FUNCTION_BLOCK TcoCvirII EXTENDS TcoCore.TcoComponent IMPLEMENTS ITcoScrewdriver //TODO: EXTENDS TcoIo.TcoPnIoComponent //IMPLEMENTS TcoAbstractions.ITcoScrewdriver
VAR_IN_OUT
	inoIoData : TcoCvirII_Io;
END_VAR

VAR
	_config : TcoCvirII_Config;
	_status : TcoCvirII_Status;
END_VAR

VAR
	_data : TcoCvirII_Data;
	_results : TcoCvirII_Results;
	
	_state : TcoCore.TcoState(THIS^, eRestoreMode.None);
	
	{attribute 'hide'}
	_timer : TON;

	//INPUT VARIABLES	
	{attribute addProperty Name "<#Screwing Program Number#>"}
	_programNo : BYTE;
	{attribute addProperty Name "<#Automatic Start#>"}
	_automaticStart : BOOL;
	
	{attribute addProperty Name "<#Run screwing cycle#>"}
	_screwingTask : TcoCore.TcoTask(THIS^);					//sequence
	
//	{attribute addProperty Name "<#Screwing program number#>"}	
//	_programNumber : BYTE; 
	{attribute addProperty Name "<#Set screwing program#>"}
	_setScrewingProgramTask : TcoCore.TcoTask(THIS^); 		//waiting for hw response
	
	{attribute addProperty Name "<#Enable#>"}
	_enableTask : TcoCore.TcoTask(THIS^);					//immediately done
	{attribute addProperty Name "<#Disable#>"}
	_disableTask : TcoCore.TcoTask(THIS^);
	{attribute addProperty Name "<#Forward#>"}
	_forwardTask : TcoCore.TcoTask(THIS^);					//sequence
	{attribute addProperty Name "<#Reverse#>"}
	_reverseTask : TcoCore.TcoTask(THIS^);					//sequence
	{attribute addProperty Name "<#Restore#>"}
    _restoreTask : TcoCore.TcoTask(THIS^);
END_VAR

VAR
    {attribute 'hide'} 
	_varInfo : __SYSTEM.VAR_INFO;
    {attribute 'hide'} 
	_sb : TcoCore.StringBuilder;
END_VAR

IF InvalidReference() THEN
    RETURN;
END_IF

//SUPER^(inPnIoBoxState := THIS^.inoIoData.PnIoBoxState, inPnIoBoxDiag := THIS^.inoIoData.PnIoBoxDiag);

InitializeComponent();

//IF NOT SUPER^.ProfinetReady THEN
//	THIS^._status.ActionDescription := '<#Not ready for operation by means of Profinet network!#>';	
//END_IF

//IF SUPER^.ProfinetReady AND THIS^._status.ActionDescription = '<#Not ready for operation by means of Profinet network!#>' THEN
//	THIS^._status.ActionDescription := '<#Ready for operation!#>';	
//END_IF

//*************RESTORE********************
_restoreTask.Enabled := TRUE;
IF _restoreTask.Execute() THEN
	Restore();
END_IF
//****************************************

//**********SET SCREWING PROGRAM**********
_setScrewingProgramTask.Enabled := TRUE;
IF _setScrewingProgramTask.Execute() THEN
	_data.ScrewingProgramOUT := _programNo;
	IF (_data.ScrewingProgramOUT  = _data.ScrewingProgramIN) THEN
		_setScrewingProgramTask.DoneWhen(TRUE);
	END_IF
END_IF
//****************************************

//****************SCREWING****************
_screwingTask.Enabled := NOT _forwardTask.Busy AND NOT _reverseTask.Busy;
IF _screwingTask.Execute() THEN
	_screwingTask.DoneWhen(ScrewingInternal());
END_IF
//****************************************

//****************ENABLE******************
_enableTask.Enabled := TRUE;
IF _enableTask.Execute() THEN
	_data.Control.SpindleValidation := TRUE;
	_enableTask.DoneWhen(TRUE);
END_IF
//****************************************

//****************DISABLE******************
_disableTask.Enabled := TRUE;
IF _disableTask.Execute() THEN
	_data.Control.SpindleValidation := FALSE;
	_disableTask.DoneWhen(TRUE);
END_IF
//*****************************************

//****************FORWARD******************
_forwardTask.Enabled := NOT _screwingTask.Busy AND NOT _reverseTask.Busy;
IF _forwardTask.Execute() THEN
	_forwardTask.DoneWhen(ScrewClockwiseInternal());
END_IF
//*****************************************

//****************REVERSE******************
_reverseTask.Enabled := NOT _screwingTask.Busy AND NOT _forwardTask.Busy;
IF _reverseTask.Execute() THEN
	_reverseTask.DoneWhen(ScrewCounterClockwiseInternal());
END_IF
//*****************************************

(*~
	<docu>
		<summary>
			Gets the configuration of the screwdriver. 					
		</summary>			
	</docu>	
~*)
PROPERTY Config : REFERENCE TO TcoCvirII_Config
GET
Config REF= _config;
END_GET
END_PROPERTY

PROPERTY DisableTask : TcoCore.ITcoTaskStatus
GET
DisableTask := THIS^._disableTask;
END_GET
END_PROPERTY

PROPERTY EnableTask : TcoCore.ITcoTaskStatus
GET
EnableTask := THIS^._enableTask;
END_GET
END_PROPERTY

PROPERTY ForwardTask : TcoCore.ITcoTaskStatus
GET
ForwardTask := THIS^._forwardTask;
END_GET
END_PROPERTY

METHOD PRIVATE InitializeComponent
VAR_INPUT
END_VAR
IF(InvalidReference()) THEN
	RETURN;
END_IF

//Reading input data
_data.Status.CycleBit1 := inoIoData.Status.0;
_data.Status.CycleBit2 := inoIoData.Status.1;
_data.Status.CycleBit4 := inoIoData.Status.2;
_data.Status.Ready := inoIoData.Status.3;
_data.Status.InCycle := inoIoData.Status.4;
_data.Status.Passed := inoIoData.Status.5;
_data.Status.Failed := inoIoData.Status.6;
_data.Status.NumberOfCyclesOk := inoIoData.Status.7;

_data.ScrewingProgramIN := inoIoData.ScrewingProgramIN;

_data.Torque := inoIoData.Torque;
_data.TorqueTrend := inoIoData.TorqueTrend;
_data.Angle := inoIoData.Angle;
_data.AngleTrend := inoIoData.AngleTrend;


//Write output data
inoIoData.Control.0 := _data.Control.CycleBit1;
inoIoData.Control.1 := _data.Control.CycleBit2;
inoIoData.Control.2 := _data.Control.CycleBit4;
inoIoData.Control.3 := _data.Control.SpindleValidation;
inoIoData.Control.4 := _data.Control.ErrorAck;
inoIoData.Control.5 := _data.Control.StartCycle;
inoIoData.Control.6 := _data.Control.Direction;
inoIoData.Control.7 := _data.Control.Reset;

inoIoData.ScrewingProgramOUT := _data.ScrewingProgramOUT;
END_METHOD

METHOD INTERNAL InvalidReference : BOOL
InvalidReference := FALSE;
IF NOT __ISVALIDREF(inoIoData) THEN
	_varInfo :=__VARINFO(inoIoData);
	Messenger.Error(_sb.Clear().Append('<#Invalid reference: #>').Append(_varInfo.Symbol).ToString());
    InvalidReference := TRUE;
END_IF
END_METHOD

(*~
	<docu>
		<summary>
			Restores this instance to the Ready state. Can be called explicitly or from within one of the restore mechanisms.	
		</summary>			
	</docu>	
~*)
METHOD  Restore : ITcoRestorable
_screwingTask.Restore();
_setScrewingProgramTask.Restore();

_enableTask.Restore();
_disableTask.Restore();

_forwardTask.Restore();
_reverseTask.Restore();

_state.Restore();

THIS^._results.Torque := 0;
THIS^._results.TorqueTrend := 0;
THIS^._results.Angle := 0;
THIS^._results.AngleTrend := 0;
	
IF InvalidReference() THEN
    RETURN;
END_IF

Tc2_System.MEMSET(destAddr:= ADR(THIS^.inoIoData) , fillByte:= 0 , n:= SIZEOF(THIS^.inoIoData));

_status.ActionDescription := '<#Restore executed!#>';
_restoreTask.Restore();
END_METHOD

PROPERTY Results : TcoCvirII_Results
GET
Results := _results;
END_GET
END_PROPERTY

PROPERTY ReverseTask : TcoCore.ITcoTaskStatus
GET
ReverseTask := THIS^._reverseTask;
END_GET
END_PROPERTY

METHOD ScrewClockwise : TcoCore.ITcoTaskStatus
VAR_INPUT
	AutomaticStart : BOOL;
END_VAR
_automaticStart := AutomaticStart;
ScrewClockwise := THIS^._forwardTask.Invoke();
END_METHOD

METHOD INTERNAL ScrewClockwiseInternal : BOOL
ScrewClockwiseInternal := FALSE;

IF (InvalidReference()) THEN
	RETURN;
END_IF

IF (_state.State<0) THEN
	_state.ChangeState(0);
END_IF

//Initialization	
IF (_state.State=0) THEN
	_state.ChangeState(30);
END_IF

//Waiting for device ready	
IF (_state.State=30) THEN
	IF _data.Status.Ready THEN
		_state.ChangeState(40);
	END_IF
END_IF

//Start cycle	
IF (_state.State=40) THEN
	_data.Control.Direction := FALSE;
	//_data.Control.SpindleValidation := TRUE;
	_data.Control.StartCycle := _automaticStart;
	IF _data.Status.InCycle THEN
		_state.ChangeState(50);
	END_IF
END_IF

//Done
IF (_state.State=50) THEN
	_state.Restore();
	ScrewClockwiseInternal := TRUE;
END_IF
END_METHOD

METHOD ScrewCounterClockwise : TcoCore.ITcoTaskStatus
VAR_INPUT
	AutomaticStart : BOOL;
END_VAR
_automaticStart := AutomaticStart;
ScrewCounterClockwise := THIS^._reverseTask.Invoke();
END_METHOD

METHOD INTERNAL ScrewCounterClockwiseInternal : BOOL
ScrewCounterClockwiseInternal := FALSE;

IF(InvalidReference()) THEN
	RETURN;
END_IF

IF (_state.State<0) THEN
	_state.ChangeState(0);
END_IF

//Initialization
IF (_state.State=0) THEN
	_state.ChangeState(40);
END_IF

//Waiting for device ready
IF (_state.State=40) THEN
	IF _data.Status.Ready THEN
		_state.ChangeState(50);
	END_IF
END_IF

//Start cycle
IF (_state.State=50) THEN
	_data.Control.Direction := TRUE;
	//_data.Control.SpindleValidation := TRUE;
	_data.Control.StartCycle := _automaticStart;
	IF _data.Status.InCycle THEN
		_state.ChangeState(60);
	END_IF
END_IF

//Done
IF (_state.State=60) THEN
	_state.Restore();	
	ScrewCounterClockwiseInternal := TRUE;
END_IF
END_METHOD

METHOD Screwing : TcoCore.ITcoTaskStatus
VAR_INPUT
	ProgramNo : BYTE;
END_VAR
_programNo := ProgramNo;
_automaticStart := TRUE;
Screwing := THIS^._screwingTask.Invoke();
END_METHOD

METHOD INTERNAL ScrewingInternal : BOOL
IF (InvalidReference()) THEN
	RETURN;
END_IF

ScrewingInternal := FALSE;

IF (_state.State<0) THEN
	_state.ChangeState(0);
END_IF

//Initialization
IF (_state.State=0) THEN
	_state.ChangeState(10);
END_IF

//Set screwing program
IF (_state.State=10) THEN
	_data.ScrewingProgramOUT := _programNo;
	IF (_data.ScrewingProgramOUT  = _data.ScrewingProgramIN) THEN
		_state.ChangeState(20);
	END_IF

	THIS^.Messenger.Debug('Set screwing program.');
END_IF

//Check screwdriver ready
IF (_state.State=20) THEN
	_timer(IN := TRUE, PT := T#2S);
	
	THIS^._data.Control.SpindleValidation := TRUE;
	
	IF THIS^._data.Status.Ready THEN
		_state.ChangeState(30);
	END_IF

	IF NOT THIS^._data.Status.Ready AND _timer.Q THEN
		THIS^.Messenger.Warning('<#Screwdriver not ready.#>');
	END_IF
END_IF

//Check screwdriver started
IF (_state.State=30) THEN
	_timer(IN := TRUE, PT := T#2S);
	
	_data.Control.Direction := FALSE;
	//_data.Control.SpindleValidation := TRUE;
	_data.Control.StartCycle := _automaticStart;
	IF _data.Status.InCycle THEN
		_timer(IN:=FALSE);
		_state.ChangeState(40);
	ELSIF _automaticStart AND NOT THIS^._data.status.InCycle AND _timer.Q THEN
		THIS^.Messenger.Debug('Screwdriver not started.');
	END_IF
END_IF

//Check screwdriver finished
IF (_state.State=40) THEN
	_timer(IN := TRUE, PT := T#2S);
	IF NOT THIS^._data.Status.InCycle THEN
		_timer(IN:=FALSE);
		_state.ChangeState(60);
	ELSIF THIS^._data.Status.InCycle AND _timer.Q THEN
		THIS^.Messenger.Debug('Screwdriver not finished.');
	END_IF
END_IF

//Reset StartCycle signal
IF (_state.State=60) THEN
	THIS^._data.Control.StartCycle := FALSE;
	_data.Control.SpindleValidation := FALSE;
	_state.ChangeState(70);
END_IF

//Collect result data
IF (_state.State=70) THEN
	THIS^._results.Angle := THIS^._data.Angle;
	THIS^._results.AngleTrend := THIS^._data.AngleTrend;
	THIS^._results.Torque := THIS^._data.Torque;
	THIS^._results.TorqueTrend := THIS^._data.TorqueTrend;
	_state.ChangeState(80);
END_IF

//Done
IF (_state.State=80) THEN
	_state.Restore();
	ScrewingInternal :=TRUE;
END_IF
END_METHOD

PROPERTY ScrewingTask : TcoCore.ITcoTaskStatus
GET
ScrewingTask := THIS^._screwingTask;
END_GET
END_PROPERTY

METHOD ScrewingWithAutomaticStart : TcoCore.ITcoTaskStatus
VAR_INPUT
	ProgramNo : BYTE;
	AutomaticStart : BOOL;
END_VAR
_programNo := ProgramNo;
_automaticStart := AutomaticStart;
ScrewingWithAutomaticStart := THIS^._screwingTask.Invoke();
END_METHOD

(*~
	<docu>
		<summary>
		    Custom service (manual, maintenance) logic.
			This method must be implemented in derived class.
		</summary>			
	</docu>	
~*)
METHOD PROTECTED  ServiceMode
END_METHOD

PROPERTY SetScrewingProgramTask : TcoCore.ITcoTaskStatus
GET
SetScrewingProgramTask := THIS^._setScrewingProgramTask;
END_GET
END_PROPERTY

(*~
	<docu>
		<summary>
			Gets the status of the screwdriver. 					
		</summary>			
	</docu>	
~*)
PROPERTY Status : REFERENCE TO TcoCvirII_Status
GET
Status REF= _status;
END_GET
END_PROPERTY

END_FUNCTION_BLOCK

(* stored: Version 1.1.0.1
   POU TcoCvirII: Id {c305f929-a2d4-40de-88d1-0f089dc5dd68}, SpecialFunc None
   Folder _Internals: Id {15bb9f30-74ce-4a79-904b-d6d9cf546a32}
   Folder Operations: Id {efcda785-c2ff-4f3c-8ac5-4fae255d743d}
   Folder Tasks: Id {4caea513-dbf2-4fc6-a892-0214b0d0def2}
   Property Config: Id {d097aa82-3255-4848-8d04-863bfbd6ce53}
   Get Get: Id {f0a60fa8-c67f-4d62-a6b9-546c59aac019}
   Property DisableTask: Id {8088f83d-5719-4515-a225-9987cf2b6650}
   Get Get: Id {994090bc-6ae9-4d0c-8c10-5634587748e7}
   Property EnableTask: Id {605e007d-c265-4186-b55e-0f3135a348ff}
   Get Get: Id {03382cd9-641c-408a-af3f-b3c52bb03cf0}
   Property ForwardTask: Id {48d179b9-4550-4ff6-9512-5ff84db8b04c}
   Get Get: Id {a80d4c0f-c000-42fb-9854-f4fcbbe19df8}
   Method InitializeComponent: Id {1c5e9459-c3a5-4faa-93ef-1c1b9a05397b}
   Method InvalidReference: Id {3fb9cd7d-6da0-44fd-8dad-f3fee2f03612}
   Method Restore: Id {b59bc427-e777-423a-b569-9ea0401f7842}
   Property Results: Id {0dc966e9-0758-48f9-94ae-403d475eecf0}
   Get Get: Id {a6751168-99e6-4edd-be02-22276c6b2605}
   Property ReverseTask: Id {8afef5ce-b48f-4540-b571-de4f4649d570}
   Get Get: Id {2e94ebca-508a-48d7-9c7e-83d3edff2f95}
   Method ScrewClockwise: Id {17a4fe0f-cbdb-44b8-b61e-b1d28e5474f6}
   Method ScrewClockwiseInternal: Id {12b8b5a9-e646-4bcd-b1f2-cad2ebce7ff3}
   Method ScrewCounterClockwise: Id {17774663-1986-4eef-9c98-4bedf4780ad5}
   Method ScrewCounterClockwiseInternal: Id {2b9f336f-e584-45b1-9583-92dcfb6afc59}
   Method Screwing: Id {376db3da-4c91-437e-b2da-76af7fb6fa76}
   Method ScrewingInternal: Id {1b5cb66f-49ef-465b-b4bc-8643a6ff9746}
   Property ScrewingTask: Id {7cc4d045-588e-4533-a5bf-32b3ff2c207e}
   Get Get: Id {f0c26b60-1844-44bf-abe4-13a0d740cf76}
   Method ScrewingWithAutomaticStart: Id {54b738e3-f415-43be-80e7-1b2dde8e49cd}
   Method ServiceMode: Id {b30ae61c-6cb6-4c11-b997-c67bc593c5c6}
   Property SetScrewingProgramTask: Id {6a502898-a737-4abe-9c46-c5a298c2cbad}
   Get Get: Id {44ae92ef-8c11-455b-b83c-33b045ec5189}
   Property Status: Id {9f04587f-2cd5-4ce7-965a-55ffcb50b2dd}
   Get Get: Id {a5b8a1d1-9db9-4d07-bddd-cbac49d95ee9} *)
